INTERFACE ICollisionGroup

METHOD Disable : BOOL
VAR_INPUT
END_VAR
END_METHOD

METHOD Enable : BOOL
VAR_INPUT
END_VAR
END_METHOD

PROPERTY GroupRef : reference to AXES_GROUP_REF
GET
END_GET
END_PROPERTY

PROPERTY GroupState : CAGroupStatus
GET
END_GET
END_PROPERTY

METHOD Reset : BOOL
VAR_INPUT
END_VAR
END_METHOD

END_INTERFACE

(* stored: Version 1.1.0.1, ProductVersion 3.1.4024.12
   Itf ICollisionGroup: Id {3fc566cf-3f15-4187-97a8-f8d156c2ea05}
   Method Disable: Id {716927af-8c3f-479d-962f-20b060f08214}
   Method Enable: Id {7961c446-8ffb-4a93-bee2-efac793ad03b}
   Property GroupRef: Id {da70f768-e857-4f18-9014-1c57ab869df0}
   Get Get: Id {ff65d9fd-a0fb-4014-a5bd-11ea974f60f4}
   Property GroupState: Id {ccaa4875-e7b8-4aad-9434-8ae988f5aafa}
   Get Get: Id {6ce504cb-b674-4e50-8b81-3854a9614761}
   Method Reset: Id {52cfbceb-29c1-48af-b76e-6022383fab33} *)
